FUNCTION_BLOCK TransportSequence EXTENDS ZApplication.Sequence
VAR
  {attribute 'hide'}
  _parent : REFERENCE TO TransportUnit;
  _io : REFERENCE TO TransportIo;
  _actuator : REFERENCE TO TransportActuator;
  _fieldbus : REFERENCE TO TransportFieldbus;
  _axis : REFERENCE TO TransportAxis;
  _data : REFERENCE TO TransportDataRef;
  _unit : REFERENCE TO TransportLinkedUnit;  
END_VAR

METHOD FB_init : BOOL
VAR_INPUT
  bInitRetains : BOOL; // if TRUE, the retain variables are initialized (warm start / cold start)
  bInCopyCode : BOOL;  // if TRUE, the instance afterwards gets moved into the copy code (online change)
  unit : REFERENCE TO TransportUnit;
END_VAR
_parent REF= unit;
_alarming := unit._alarming;
_io REF= unit._equipment.Io;
_actuator REF= unit._equipment.Actuator;
_fieldbus REF= unit._equipment.Fieldbus;
_axis REF= unit._equipment.Axis;
_unit REF= unit._equipment.Unit;
_data REF= unit._data;
_loggerDiagnostics.SetLogger(unit._logger);
END_METHOD

METHOD StepDecoded : ZCore.ZString
VAR_INPUT
  stepIndex : INT;
END_VAR
VAR_INST
  _stepIndexDecoded : TransportStep;
END_VAR
_stepIndexDecoded := stepIndex;
stepDecoded := TO_STRING(_stepIndexDecoded);
END_METHOD

END_FUNCTION_BLOCK

(* stored: Version 1.1.0.1
   POU TransportSequence: Id {7ab3c77b-32e1-4578-a881-73c26a71e1c0}, SpecialFunc None
   Method FB_init: Id {7eb91854-a8a3-4af0-8313-6016c3190fa5}
   Method StepDecoded: Id {e26d5f97-ce8e-4e3b-81be-a7ae27b195da} *)
